// TIA Portal project "Lab1.3" (V16)

(* hardware
DEVICE "S7-1200 station_1"  S7-1200 Station
   slot 0: "Rack_0"  S7-1200 Rack  Rack  V1.0
   slot 1: "PLC_1"  CPU 1211C AC/DC/Rly  6ES7 211-1BE40-0XB0  V4.4
DEVICE "HMI_1"  KTP700 Basic PN
   slot 0: "HMI_1"  KTP700 Basic PN  6AV2 123-2GB03-0AX0  16.0.0.0
   slot 1: "HMI_RT_1"  KTP700 Basic PN  6AV2 123-2GB03-0AX0  16.0.0.0
   slot 5: "HMI_1.IE_CP_1"  PROFINET Interface  16.0.0.0
      slot 1: "PROFINET Interface_1"  PROFINET Interface
         slot 1: "Port_1"  Port
DEVICE "HMI_2"  KTP700 Basic PN
   slot 0: "HMI_2"  KTP700 Basic PN  6AV2 123-2GB03-0AX0  15.1.0.0
   slot 1: "HMI_RT_2"  KTP700 Basic PN  6AV2 123-2GB03-0AX0  15.1.0.0
   slot 5: "HMI_2.IE_CP_1"  PROFINET Interface  15.0.1.0
      slot 1: "PROFINET Interface_1"  PROFINET Interface
         slot 1: "Port_1"  Port
*)

// ===== PLC "PLC_1"  CPU 1211C AC/DC/Rly =====

VAR_GLOBAL   // PLC tag table "Default tag table"
   "LAMP_1" AT %Q0.0 : Bool;   // Đèn 1 xanh
   "LAMP_2" AT %Q0.1 : Bool;   // Đèn 2 vàng
   "START" AT %M0.3 : Bool;   // Nút START
   "STOP" AT %M0.0 : Bool;   // Nút STOP
   "SIG_SCAN" AT %M0.2 : Bool;   // Bộ nhớ scan L2
   "RESET_TAG" AT %M0.1 : Bool;   // Tự reset CTU
   "COUNTER_INPUT" AT %MW100 : Int;   // Giới hạn N
   "COUNTER_DISPLAY" AT %MW26 : Int;   // Giá trị đếm CV
   "T1_INPUT" AT %MD200 : DInt;   // Thời gian T1 nhập
   "T1_RESULT" AT %MD6 : DInt;   // T1 × 1000 ms
   "T2_INPUT" AT %MD10 : DInt;   // Thời gian T2 nhập
   "T2_RESULT" AT %MD14 : DInt;   // T2 × 1000 ms
   "T1_HMI" AT %MD18 : DInt;   // Hiển thị T1 elapsed
   "T2_HMI" AT %MD22 : DInt;   // Hiển thị T2 elapsed
   "START_P" AT %M5.0 : Bool;
END_VAR

// folder: System blocks/Program resources

DATA_BLOCK "Timer2"   // DB1
{ S7_Optimized_Access := 'TRUE' }
AUTHOR : Simatic
FAMILY : IEC
NAME : IEC_TMR
VERSION : 1.0
// stored: InstanceOfName IEC_TIMER
"IEC_TIMER"
BEGIN
END_DATA_BLOCK

DATA_BLOCK "Timer1"   // DB2
{ S7_Optimized_Access := 'TRUE' }
AUTHOR : Simatic
FAMILY : IEC
NAME : IEC_TMR
VERSION : 1.0
// stored: InstanceOfName IEC_TIMER
"IEC_TIMER"
BEGIN
END_DATA_BLOCK

DATA_BLOCK "COUNTER"   // DB3
{ S7_Optimized_Access := 'TRUE' }
AUTHOR : Simatic
FAMILY : IEC
NAME : CNTR
VERSION : 1.0
// stored: InstanceOfName IEC_COUNTER
"IEC_COUNTER"
BEGIN
END_DATA_BLOCK

DATA_BLOCK "RESET_DELAY"   // DB4
{ S7_Optimized_Access := 'TRUE' }
AUTHOR : Simatic
FAMILY : IEC
NAME : IEC_TMR
VERSION : 1.0
// stored: InstanceOfName IEC_TIMER
"IEC_TIMER"
BEGIN
END_DATA_BLOCK

// folder: (top level)

ORGANIZATION_BLOCK "Main"   // OB1, LAD, ProgramCycle
TITLE = "Main Program Sweep (Cycle)"
{ S7_Optimized_Access := 'TRUE' }
VERSION : 0.1
   VAR_INPUT
      Initial_Call : Bool;   // Initial call of this OB
      Remanence : Bool;   // =True, if remanent data are available
   END_VAR
   VAR_TEMP   // added for the SCL form of the ladder/FBD networks
      _w1 : Bool;
   END_VAR
BEGIN

REGION Network 1: Đèn 1 xanh
   // START + tính PT
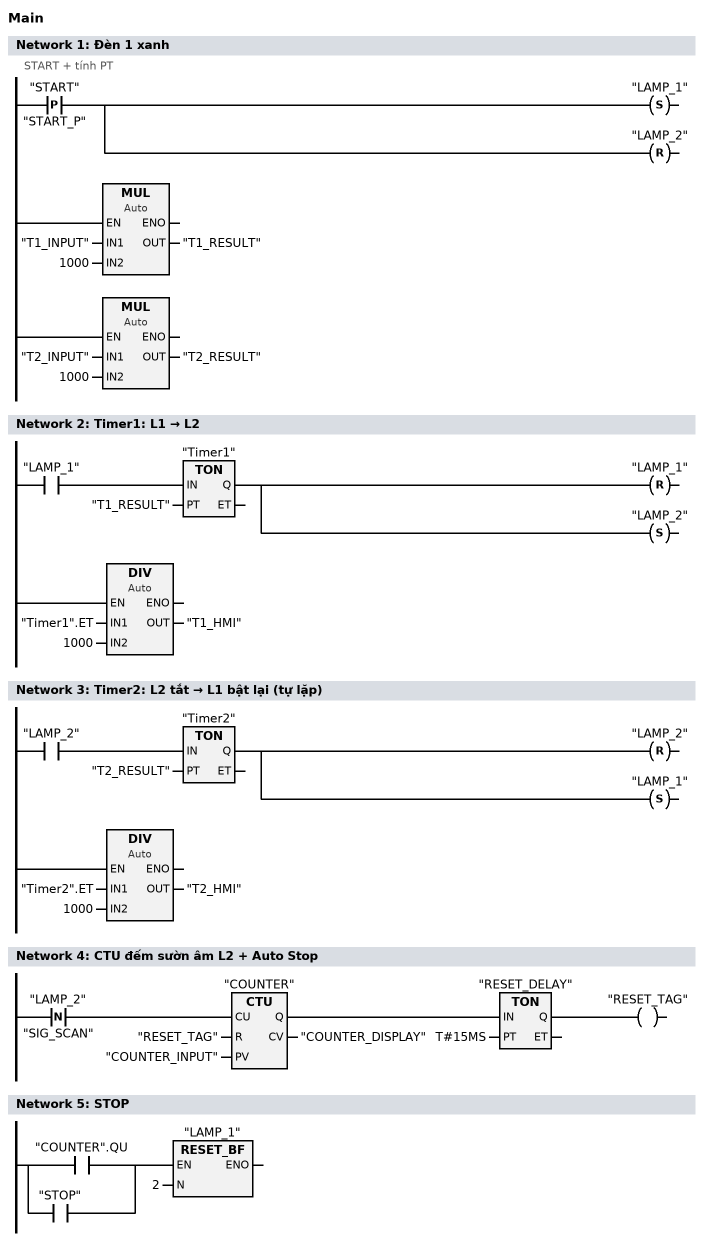
   RUNG wire#powerrail
      P_Contact(operand := "START", bit := "START_P")
      wire#w1
      S_Coil( "LAMP_1" )
   END_RUNG
   RUNG wire#w1
      R_Coil( "LAMP_2" )
   END_RUNG
   RUNG wire#powerrail
      Mul(in1 := "T1_INPUT", in2 := 1000, out => "T1_RESULT")
   END_RUNG
   RUNG wire#powerrail
      Mul(in1 := "T2_INPUT", in2 := 1000, out => "T2_RESULT")
   END_RUNG
   // the same network as SCL:
   #_w1 := "START" AND NOT "START_P";   // rising edge of "START"
   "START_P" := "START";
   IF #_w1 THEN
       "LAMP_1" := TRUE;
       "LAMP_2" := FALSE;
   END_IF;
   "T1_RESULT" := "T1_INPUT" * 1000;
   "T2_RESULT" := "T2_INPUT" * 1000;
END_REGION

REGION Network 2: Timer1: L1 → L2
   "Timer1".TON(IN := "LAMP_1", PT := "T1_RESULT");
   IF "Timer1".Q THEN
       "LAMP_1" := FALSE;
       "LAMP_2" := TRUE;
   END_IF;
   "T1_HMI" := "Timer1".ET / 1000;
END_REGION

REGION Network 3: Timer2: L2 tắt → L1 bật lại (tự lặp)
   "Timer2".TON(IN := "LAMP_2", PT := "T2_RESULT");
   IF "Timer2".Q THEN
       "LAMP_2" := FALSE;
       "LAMP_1" := TRUE;
   END_IF;
   "T2_HMI" := "Timer2".ET / 1000;
END_REGION

REGION Network 4: CTU đếm sườn âm L2 + Auto Stop
   #_w1 := NOT "LAMP_2" AND "SIG_SCAN";   // falling edge of "LAMP_2"
   "SIG_SCAN" := "LAMP_2";
   "COUNTER".CTU(CU := #_w1, R := "RESET_TAG", PV := "COUNTER_INPUT", CV => "COUNTER_DISPLAY");
   "RESET_DELAY".TON(IN := "COUNTER".Q, PT := T#15MS);
   "RESET_TAG" := "RESET_DELAY".Q;
END_REGION

REGION Network 5: STOP
   // no SCL statement known for RBitfield: written as a call
   IF "COUNTER".QU OR "STOP" THEN RESET_BF(operand := "LAMP_1", n := 2); END_IF;
END_REGION
END_ORGANIZATION_BLOCK

(* ===== HMI "HMI_RT_1" =====
system functions are stored by id; their names below are inferred from use
connection "HMI_Connection_1": ETHERNET, SMART_S7_1200_OMS

HMI tags "Default tag table"
   "START" : Bool = PLC START AT %M0.3, 1 s
   "STOP" : Bool = PLC STOP AT %M0.0, 1 s
   "LAMP_1" : Bool = PLC LAMP_1 AT %Q0.0, 1 s
   "LAMP_2" : Bool = PLC LAMP_2 AT %Q0.1, 1 s
   "COUNTER_INPUT" : Int = PLC COUNTER_INPUT AT %MW100, 1 s
   "COUNTER_DISPLAY" : Int = PLC COUNTER_DISPLAY AT %MW26, 1 s
   "T1_INPUT" : DInt = PLC T1_INPUT AT %MD200, 1 s
   "T1_HMI" : DInt = PLC T1_HMI AT %MD18, 1 s
   "T2_INPUT" : DInt = PLC T2_INPUT AT %MD10, 1 s
   "T2_HMI" : DInt = PLC T2_HMI AT %MD22, 1 s

screen "Root screen" 800x480, template "Template_1"
   Button "HmiScreenItemData_1" at 36,36 size 159x47; TextOff 'System screens'; PictureOff "Navigates to System screens for KTP700 Basic+ PN 16.0.0.0"; PictureOn "Navigates to System screens for KTP700 Basic+ PN 16.0.0.0"
      on Release: ActivateScreen("System screens", 0)
   Button "Button_1" at 80,106 size 96x32; TextOff 'START'
      on Press: SetBit("START")
      on Release: ResetBit("START")
   Button "Button_2" at 80,147 size 96x32; TextOff 'STOP'
      on Press: SetBit("STOP")
      on Release: ResetBit("STOP")
   Circle "Circle_1" at 219,106 size 70x70
      Appearance <- "LAMP_1"
   Circle "Circle_2" at 337,109 size 70x70
      Appearance <- "LAMP_2"
   TextField "Text field_1" at 93,202 size 119x23; Text 'Counter Input'
   TextField "Text field_2" at 340,202 size 58x23; Text 'Count'
   IOField "I/O field_1" at 98,227 size 96x32; FormatPattern s99999
      Appearance <- "COUNTER_INPUT"
      ProcessValue <- "COUNTER_INPUT"
   IOField "I/O field_2" at 337,228 size 96x32; FormatPattern s99999
      ProcessValue <- "COUNTER_DISPLAY"
   IOField "I/O field_3" at 99,306 size 96x32; FormatPattern s9999999999
      ProcessValue <- "T1_INPUT"
   IOField "I/O field_4" at 338,307 size 96x32; FormatPattern s9999999999
      ProcessValue <- "T1_HMI"
   TextField "Text field_3" at 101,277 size 68x23; Text 'Timer 1'
   TextField "Text field_4" at 348,277 size 68x23; Text 'Elapsed'
   IOField "I/O field_5" at 101,384 size 96x32; FormatPattern s9999999999
      ProcessValue <- "T2_INPUT"
   IOField "I/O field_6" at 340,385 size 96x32; FormatPattern s9999999999
      ProcessValue <- "T2_HMI"
   TextField "Text field_5" at 103,355 size 68x23; Text 'Timer 2'
   TextField "Text field_6" at 350,355 size 68x23; Text 'Elapsed'

screen "System screens" 800x480, template "Template_1"
   Button "Back" at 1,1 size 159x47; TextOff 'Back'
      on Release: ActivateScreen("Root screen", 0)
   Button "HmiScreenItemData" at 36,95 size 159x47; TextOff 'SIMATIC PLC system diagnos...'; PictureOff "Navigates to SIMATIC PLC system diagnostics for KTP700 Basic+ PN 16.0.0.0"; PictureOn "Navigates to SIMATIC PLC system diagnostics for KTP700 Basic+ PN 16.0.0.0"
      on Release: ActivateScreen("SIMATIC PLC system diagnostics", 0)
   Button "HmiScreenItemData_1" at 36,154 size 159x47; TextOff 'Project information'; PictureOff "Navigates to Project information for KTP700 Basic+ PN 16.0.0.0"; PictureOn "Navigates to Project information for KTP700 Basic+ PN 16.0.0.0"
      on Release: ActivateScreen("Project information", 0)
   Button "HmiScreenItemData_2" at 36,213 size 159x47; TextOff 'User administration'; PictureOff "Navigates to User administration for KTP700 Basic+ PN 16.0.0.0"; PictureOn "Navigates to User administration for KTP700 Basic+ PN 16.0.0.0"
      on Release: ActivateScreen("User administration", 0)
   Button "HmiScreenItemData_3" at 36,272 size 159x47; TextOff 'System information'; PictureOff "Navigates to System information for KTP700 Basic+ PN 16.0.0.0"; PictureOn "Navigates to System information for KTP700 Basic+ PN 16.0.0.0"
      on Release: ActivateScreen("System information", 0)
   Button "HmiScreenItemData_4" at 36,331 size 159x47; TextOff 'Different jobs'; PictureOff "Navigates to Different jobs for KTP700 Basic+ PN 16.0.0.0"; PictureOn "Navigates to Different jobs for KTP700 Basic+ PN 16.0.0.0"
      on Release: ActivateScreen("Different jobs", 0)

screen "SIMATIC PLC system diagnostics" 800x480, template "Template_1"
   SysDiagControl "HmiScreenItemData" at 1,49 size 796x423
   Button "Back" at 1,1 size 159x47; TextOff 'Back'
      on Release: ActivateScreen("System screens", 0)

screen "Project information" 800x480, template "Template_1"
   TextField "HmiScreenItemData" at 35,51 size 171x28; Text 'Project name:'
   TextField "HmiScreenItemData_1" at 241,51 size 524x28; Text 'Lab1.3'
   TextField "HmiScreenItemData_2" at 35,81 size 171x28; Text 'Created on:'
   TextField "HmiScreenItemData_3" at 241,81 size 524x28; Text '6/8/2026 6:55:18 PM'
   TextField "HmiScreenItemData_4" at 35,111 size 171x28; Text 'Author:'
   TextField "HmiScreenItemData_5" at 241,111 size 524x28; Text 'Khoa'
   TextField "HmiScreenItemData_6" at 35,141 size 171x28; Text 'Description:'
   TextField "HmiScreenItemData_7" at 241,141 size 524x28; Text '(not configured)'
   Button "Back" at 1,1 size 159x47; TextOff 'Back'
      on Release: ActivateScreen("System screens", 0)

screen "User administration" 800x480, template "Template_1"
   UserView "HmiScreenItemData" at 1,49 size 796x423
   Button "Back" at 1,1 size 159x47; TextOff 'Back'
      on Release: ActivateScreen("System screens", 0)

screen "System information" 800x480, template "Template_1"
   TextField "HmiScreenItemData" at 35,51 size 171x28; Text 'HMI device type:'
   TextField "HmiScreenItemData_1" at 241,51 size 524x28; Text 'KTP700 Basic+ PN 16.0.0.0'
   TextField "HmiScreenItemData_2" at 35,81 size 171x28; Text 'Connection:'
   TextField "HmiScreenItemData_3" at 241,81 size 524x28; Text 'PROFINET (X1)'
   TextField "HmiScreenItemData_4" at 35,111 size 171x28; Text 'PLC:'
   TextField "HmiScreenItemData_5" at 241,111 size 524x28; Text 'SIMATIC S7 1200'
   Button "Back" at 1,1 size 159x47; TextOff 'Back'
      on Release: ActivateScreen("System screens", 0)

screen "Different jobs" 800x480, template "Template_1"
   Button "Online" at 36,95 size 159x47; TextOff 'Online'
      on Release: function_bb44b551(0)
   Button "Offline" at 36,154 size 159x47; TextOff 'Offline'
      on Release: function_bb44b551(1)
   Button "Transfer" at 36,213 size 159x47; TextOff 'Transfer'
      on Release: function_bb44b551(2)
   Button "Toggle language" at 36,272 size 159x47; TextOff 'Toggle language'
      on Release: function_fb9197e8(-1)
   Button "Stop Runtime" at 36,331 size 159x47; TextOff 'Stop Runtime'
      on Release: StopRuntime(0)
   Button "Back" at 1,1 size 159x47; TextOff 'Back'
      on Release: ActivateScreen("System screens", 0)
*)

(* ===== HMI "HMI_RT_2" =====
system functions are stored by id; their names below are inferred from use
connection "HMI_Connection_2": ETHERNET, SMART_S7_1200_OMS
connection "HMI_Connection_3": ETHERNET, SMART_S7_1200_OMS

HMI tags "Default tag table"
   "LAMP_1" : Bool = PLC LAMP_1 AT %Q0.0, 1 s
   "LAMP_2" : Bool = PLC LAMP_2 AT %Q0.1, 1 s
   "START" : Bool = PLC START AT %M0.3, 1 s
   "STOP" : Bool = PLC STOP AT %M0.0, 1 s
   "SIG_SCAN" : Bool = PLC SIG_SCAN AT %M0.2, 1 s
   "RESET_TAG" : Bool = PLC RESET_TAG AT %M0.1, 1 s
   "COUNTER_INPUT" : Int = PLC COUNTER_INPUT AT %MW100, 1 s
   "COUNTER_DISPLAY" : Int = PLC COUNTER_DISPLAY AT %MW26, 1 s
   "T1_INPUT" : DInt = PLC T1_INPUT AT %MD200, 1 s
   "T1_RESULT" : DInt = PLC T1_RESULT AT %MD6, 1 s
   "T2_INPUT" : DInt = PLC T2_INPUT AT %MD10, 1 s
   "T2_RESULT" : DInt = PLC T2_RESULT AT %MD14, 1 s
   "T1_HMI" : DInt = PLC T1_HMI AT %MD18, 1 s
   "T2_HMI" : DInt = PLC T2_HMI AT %MD22, 1 s
   "START_P" : Bool = PLC START_P AT %M5.0, 1 s

screen "Root screen" 800x480, template "Template_1"
   TextField "HmiScreenItemData" at 80,225 size 640x25; Text 'Welcome to HMI_2 (KTP700 Basic+ PN)!'
   Button "HmiScreenItemData_1" at 36,36 size 159x47; TextOff 'System screens'; PictureOff "Navigates to System screens for KTP700 Basic+ PN 15.1.0.0"; PictureOn "Navigates to System screens for KTP700 Basic+ PN 15.1.0.0"
      on Release: ActivateScreen("System screens", 0)
   Button "Button_1" at 80,106 size 96x32; TextOff 'START'
      on Release: ResetBit("START")
      on Press: SetBit("START")
   Button "Button_2" at 80,147 size 96x32; TextOff 'STOP'
      on Release: ResetBit("STOP")
      on Press: SetBit("STOP")
   Circle "Circle_1" at 219,106 size 70x70
      Appearance <- "LAMP_1"
   Circle "Circle_2" at 337,109 size 70x70
      Appearance <- "LAMP_2"
   TextField "Text field_1" at 93,202 size 119x23; Text 'Counter Input'
   TextField "Text field_2" at 340,202 size 58x23; Text 'Count'
   IOField "I/O field_1" at 98,227 size 96x32; FormatPattern s99999
      ProcessValue <- "COUNTER_INPUT"
      Appearance <- "COUNTER_INPUT"
   IOField "I/O field_2" at 337,228 size 96x32; FormatPattern s99999
      ProcessValue <- "COUNTER_DISPLAY"
   IOField "I/O field_3" at 99,306 size 96x32; FormatPattern s9999999999
      ProcessValue <- "T1_INPUT"
   IOField "I/O field_4" at 338,307 size 96x32; FormatPattern s9999999999
      ProcessValue <- "T1_HMI"
   TextField "Text field_3" at 101,277 size 68x23; Text 'Timer 1'
   TextField "Text field_4" at 348,277 size 68x23; Text 'Elapsed'
   IOField "I/O field_5" at 101,384 size 96x32; FormatPattern s9999999999
      ProcessValue <- "T2_INPUT"
   IOField "I/O field_6" at 340,385 size 96x32; FormatPattern s9999999999
      ProcessValue <- "T2_HMI"
   TextField "Text field_5" at 103,355 size 68x23; Text 'Timer 2'
   TextField "Text field_6" at 350,355 size 68x23; Text 'Elapsed'

screen "System screens" 800x480, template "Template_1"
   Button "Back" at 1,1 size 159x47; TextOff 'Back'
      on Release: ActivateScreen("Root screen", 0)
   Button "HmiScreenItemData" at 36,95 size 159x47; TextOff 'SIMATIC PLC system diagnos...'; PictureOff "Navigates to SIMATIC PLC system diagnostics for KTP700 Basic+ PN 15.1.0.0"; PictureOn "Navigates to SIMATIC PLC system diagnostics for KTP700 Basic+ PN 15.1.0.0"
      on Release: ActivateScreen("SIMATIC PLC system diagnostics", 0)
   Button "HmiScreenItemData_1" at 36,154 size 159x47; TextOff 'Project information'; PictureOff "Navigates to Project information for KTP700 Basic+ PN 15.1.0.0"; PictureOn "Navigates to Project information for KTP700 Basic+ PN 15.1.0.0"
      on Release: ActivateScreen("Project information", 0)
   Button "HmiScreenItemData_2" at 36,213 size 159x47; TextOff 'User administration'; PictureOff "Navigates to User administration for KTP700 Basic+ PN 15.1.0.0"; PictureOn "Navigates to User administration for KTP700 Basic+ PN 15.1.0.0"
      on Release: ActivateScreen("User administration", 0)
   Button "HmiScreenItemData_3" at 36,272 size 159x47; TextOff 'System information'; PictureOff "Navigates to System information for KTP700 Basic+ PN 15.1.0.0"; PictureOn "Navigates to System information for KTP700 Basic+ PN 15.1.0.0"
      on Release: ActivateScreen("System information", 0)
   Button "HmiScreenItemData_4" at 36,331 size 159x47; TextOff 'Different jobs'; PictureOff "Navigates to Different jobs for KTP700 Basic+ PN 15.1.0.0"; PictureOn "Navigates to Different jobs for KTP700 Basic+ PN 15.1.0.0"
      on Release: ActivateScreen("Different jobs", 0)

screen "SIMATIC PLC system diagnostics" 800x480, template "Template_1"
   SysDiagControl "HmiScreenItemData" at 1,49 size 796x423
   Button "Back" at 1,1 size 159x47; TextOff 'Back'
      on Release: ActivateScreen("System screens", 0)

screen "Project information" 800x480, template "Template_1"
   TextField "HmiScreenItemData" at 35,51 size 171x28; Text 'Project name:'
   TextField "HmiScreenItemData_1" at 241,51 size 524x28; Text 'Lab1.3'
   TextField "HmiScreenItemData_2" at 35,81 size 171x28; Text 'Created on:'
   TextField "HmiScreenItemData_3" at 241,81 size 524x28; Text '6/8/2026 6:55:18 PM'
   TextField "HmiScreenItemData_4" at 35,111 size 171x28; Text 'Author:'
   TextField "HmiScreenItemData_5" at 241,111 size 524x28; Text 'Khoa'
   TextField "HmiScreenItemData_6" at 35,141 size 171x28; Text 'Description:'
   TextField "HmiScreenItemData_7" at 241,141 size 524x28; Text '(not configured)'
   Button "Back" at 1,1 size 159x47; TextOff 'Back'
      on Release: ActivateScreen("System screens", 0)

screen "User administration" 800x480, template "Template_1"
   UserView "HmiScreenItemData" at 1,49 size 796x423
   Button "Back" at 1,1 size 159x47; TextOff 'Back'
      on Release: ActivateScreen("System screens", 0)

screen "System information" 800x480, template "Template_1"
   TextField "HmiScreenItemData" at 35,51 size 171x28; Text 'HMI device type:'
   TextField "HmiScreenItemData_1" at 241,51 size 524x28; Text 'KTP700 Basic+ PN 15.1.0.0'
   TextField "HmiScreenItemData_2" at 35,81 size 171x28; Text 'Connection:'
   TextField "HmiScreenItemData_3" at 241,81 size 524x28; Text 'PROFINET (X1)'
   TextField "HmiScreenItemData_4" at 35,111 size 171x28; Text 'PLC:'
   TextField "HmiScreenItemData_5" at 241,111 size 524x28; Text 'SIMATIC S7 1200'
   Button "Back" at 1,1 size 159x47; TextOff 'Back'
      on Release: ActivateScreen("System screens", 0)

screen "Different jobs" 800x480, template "Template_1"
   Button "Online" at 36,95 size 159x47; TextOff 'Online'
      on Release: function_bb44b551(0)
   Button "Offline" at 36,154 size 159x47; TextOff 'Offline'
      on Release: function_bb44b551(1)
   Button "Transfer" at 36,213 size 159x47; TextOff 'Transfer'
      on Release: function_bb44b551(2)
   Button "Toggle language" at 36,272 size 159x47; TextOff 'Toggle language'
      on Release: function_fb9197e8(-1)
   Button "Stop Runtime" at 36,331 size 159x47; TextOff 'Stop Runtime'
      on Release: StopRuntime(0)
   Button "Back" at 1,1 size 159x47; TextOff 'Back'
      on Release: ActivateScreen("System screens", 0)
*)